# EPICS StreamDevice protocol: siteApps-725b29e158e8061764313f5708af9e46fe30c0a8/siteApps-725b29e158e8061764313f5708af9e46fe30c0a8/glassManPS/proto/glassManPS.proto
Terminator = CR;

set_value{
        out "\x01S%s";
}

get_voltage{
	out "\x01Q51";
	in "%*c%3x%*11x";
}

get_current{
        out "\x01Q51";
        in "%*c%*3x%3x%*8x";
}

get_st{
        out "\x01Q51";
        in "%*c%*9x%1x%*4x";
}

set_reset{
	out "\x01S0300000000004CA";
	in "%s";
}
